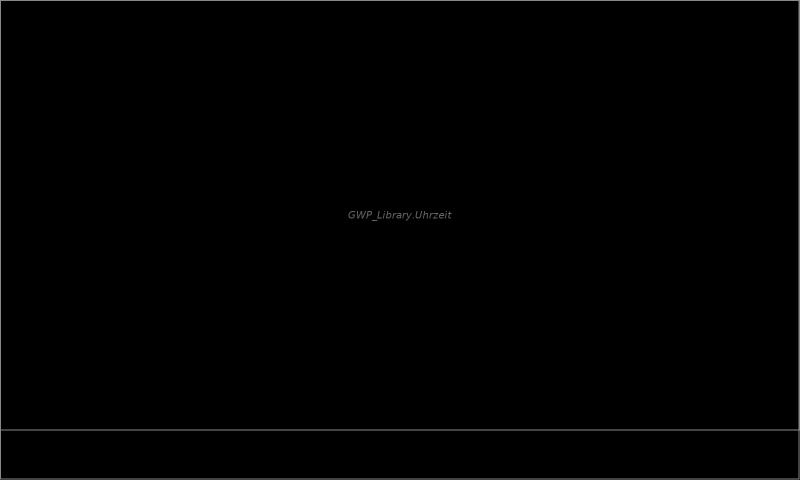
VISUALIZATION Uhr_Einstellen  // 800x480
    Frame (0,0 800x430)
        shows GWP_Library.Uhrzeit(FB_Init_1 := Main.Init_0, i_Titel := 37)
END_VISUALIZATION

(* stored: Version 1.1.0.1, ProductVersion 3.1.4022.6
   Visu Uhr_Einstellen: Id {5e67def1-e8c5-4756-a912-015c22945011} *)
